(* IEC 61131-3 sources: Industry-PLC-LLM/data/PLCBEAD_repo/PLCBEAD_PLCEmbed-main/PLC-BEAD/Source/GEB/WINDOW, 1 file *)

(* ---- WINDOW.ST ---- *)
FUNCTION WINDOW:BOOL
	VAR_INPUT
		LOW :	REAL;
		IN :	REAL;
		HIGH :	REAL;
	END_VAR
	window := (IN < high) AND (IN > LOW);

END_FUNCTION

PROGRAM program0
  	VAR
		LOW :	REAL;
		IN :	REAL;
		HIGH :	REAL;
		CEIL5_OUT : BOOL;
	END_VAR

  	CEIL5_OUT := window(LOW, IN, HIGH);
END_PROGRAM
